ABB RobotStudio station: Eksamens.rspag

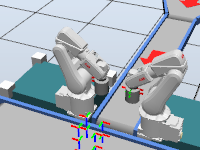
--- station ---
Station Eksamens (saved by RobotStudio 7.0.8746.631)
Controller Virtual_controller, task T_ROB3: task frame (RAPID world) sits at (-5805.06, 703.5, 890) mm, rotated rx 0 ry 0 rz -90 deg in the station
Controller Virtual_controller, task T_ROB2: task frame (RAPID world) sits at (-5805.06, 703.5, 890) mm, rotated rx 0 ry 0 rz -90 deg in the station
Controller Virtual_controller, task T_ROB1: task frame (RAPID world) sits at (-5805.06, 703.5, 890) mm, rotated rx 0 ry 0 rz -90 deg in the station
Controller Virtual_controller
  mechanical unit ROB_1: IRB120_3_58__01_2, 6 joints, base frame (83.5, -144.94, 0) mm
  mechanical unit ROB_2: IRB2600_20_165_C_01_2, 6 joints, base frame (1331.39, 3332.7, 0) mm, rotated rx 0 ry 0 rz 180 deg
  mechanical unit ROB_3: IRB120_3_58__01_3, 6 joints, base frame (643.5, -144.94, 0) mm, rotated rx 0 ry 0 rz 180 deg
Layout (positions relative to the parent item):
  - Sorter_kasser [graphiccomponentgroup]
    - Assemblies [graphiccomponentgroup]
      - Section1 [graphiccomponentgroup]
        - ABB_IRC5_ctrl [graphiccomponentgroup]
          - ABB_IRC5_ctrl_1 [graphiccomponentgroup]
            - Mesh0 [part]
        - Conveyor__Straight_ [graphiccomponentgroup]
          - CONVEYOR1 [graphiccomponentgroup]
            - Mesh1 [part]
            - Mesh2 [part]
            - Mesh3 [part]
          - CONVEYOR2 [graphiccomponentgroup]
            - Mesh4 [part]
            - Mesh5 [part]
            - Mesh6 [part]
          - CONVEYOR3 [graphiccomponentgroup]
            - Mesh7 [part]
            - Mesh8 [part]
            - Mesh9 [part]
          - CONVEYOR4 [graphiccomponentgroup]
            - Mesh10 [part]
            - Mesh11 [part]
            - Mesh12 [part]
          - CONVEYOR5 [graphiccomponentgroup]
            - Mesh13 [part]
            - Mesh14 [part]
            - Mesh15 [part]
          - CONVEYOR6 [graphiccomponentgroup]
            - Mesh16 [part]
            - Mesh17 [part]
            - Mesh18 [part]
          - CONVEYOR7 [graphiccomponentgroup]
            - Mesh19 [part]
            - Mesh20 [part]
            - Mesh21 [part]
        - Cube [graphiccomponentgroup]
          - Cube1 [graphiccomponentgroup]
            - Mesh22 [part]
            - Mesh23 [part]
            - Mesh24 [part]
            - Mesh25 [part]
            - Mesh26 [part]
          - Cube2 [graphiccomponentgroup]
            - Mesh27 [part]
            - Mesh28 [part]
            - Mesh29 [part]
            - Mesh30 [part]
            - Mesh31 [part]
          - Cube3 [graphiccomponentgroup]
            - Mesh32 [part]
            - Mesh33 [part]
            - Mesh34 [part]
            - Mesh35 [part]
            - Mesh36 [part]
        - Eater [graphiccomponentgroup]
          - EATER1 [graphiccomponentgroup]
            - Mesh37 [part]
        - Display [graphiccomponentgroup]
          - EaterSmall [graphiccomponentgroup]
            - Mesh38 [part]
            - Mesh39 [part]
            - Mesh40 [part]
            - Mesh41 [part]
            - Mesh42 [part]
            - Mesh43 [part]
            - Mesh44 [part]
            - Mesh45 [part]
            - Mesh46 [part]
            - Mesh47 [part]
            - Mesh48 [part]
        - Feeder [graphiccomponentgroup]
          - FEEDER1 [graphiccomponentgroup]
            - Mesh49 [part]
            - Mesh50 [part]
          - FEEDER2 [graphiccomponentgroup]
            - Mesh51 [part]
            - Mesh52 [part]
          - FEEDER3 [graphiccomponentgroup]
            - Mesh53 [part]
            - Mesh54 [part]
        - Scale [graphiccomponentgroup]
          - Scale_Weight [graphiccomponentgroup]
            - Mesh55 [part]
            - Mesh56 [part]
            - Mesh57 [part]
            - Mesh58 [part]
          - Scale_Weight1 [graphiccomponentgroup]
            - Mesh59 [part]
            - Mesh60 [part]
            - Mesh61 [part]
            - Mesh62 [part]
          - Scale_Weight2 [graphiccomponentgroup]
            - Mesh63 [part]
            - Mesh64 [part]
            - Mesh65 [part]
            - Mesh66 [part]
        - Text [graphiccomponentgroup]
          - Text1 [graphiccomponentgroup]
            - Mesh67 [part]
    - Motors [graphiccomponentgroup]
      - Surface [graphiccomponentgroup]
        - MOTOR1 [graphiccomponentgroup]
          - Mesh75 [part]
          - Mesh76 [part]
          - Mesh77 [part]
          - Mesh78 [part]
        - MOTOR6 [graphiccomponentgroup]
          - Mesh79 [part]
        - MOTOR8 [graphiccomponentgroup]
          - Mesh80 [part]
        - MOTOR9 [graphiccomponentgroup]
          - Mesh81 [part]
    - Loads [graphiccomponentgroup]
      - Mesh68 [part]
      - Mesh69 [part]
      - Mesh70 [part]
      - Mesh71 [part]
      - Mesh72 [part]
      - Mesh73 [part]
      - Mesh74 [part]
  - IRB120_3_58__01_2 [mechanism, from Robots\IRB120_3_58_G_01.rslib] at (-5950, 620, 890) mm, rotated rx 0 ry 0 rz -90 deg; joint values [-0.0062, -0.4744, 1.1199, 0, 0.9253, -0.0062] (rad or m)
  - IRB2600_20_165_C_01_2 [mechanism, from Robots\IRB2600_20_165_C_01.rslib] at (-2472.36, -627.89, 890) mm, rotated rx 0 ry 0 rz 90 deg; joint values [0, 0.2407, 0.4991, 6.2832, 0.831, 0] (rad or m)
  - IRB120_3_58__01_3 [mechanism, from Robots\IRB120_3_58_G_01.rslib] at (-5950, 60, 890) mm, rotated rx 0 ry 0 rz 90 deg; joint values [0.006, -0.4425, 1.1015, 0, 0.9118, 0.006] (rad or m)
  - GripperStackerRight [mechanism] at (-5951, 460, 1222.41) mm, rotated rx 180 ry 0 rz 90 deg
      TCP GripperStackerRight at (0, 0, 30) mm
      links: SimpleGripper
  - GripperStackerLeft [mechanism] at (-5951, 226, 1222.41) mm, rotated rx 180 ry 0 rz -90 deg
      TCP GripperStackerLeft at (0, 0, 30) mm
      links: SimpleGripper
  - GripperSorter [mechanism] at (-2472.36, 353.71, 1478.82) mm, rotated rx 180 ry 0 rz -90 deg
      TCP GripperSorter at (0, 0, 30) mm
      links: SimpleGripper
Attachment: GripperStackerRight is attached to IRB120_3_58__01_2 / Link6
Attachment: GripperStackerLeft is attached to IRB120_3_58__01_3 / Link6
Attachment: GripperSorter is attached to IRB2600_20_165_C_01_2 / Link6

--- Backups/Virtual_controller/RAPID/TASK1/PROGMOD/CalibData.mod ---
MODULE CalibData
	PERS tooldata GripperStackerRight:=[TRUE,[[0,0,30],[1,0,0,0]],[1,[0,0,1],[1,0,0,0],0,0,0]];
ENDMODULE

--- Backups/Virtual_controller/RAPID/TASK1/PROGMOD/Module1.mod ---
MODULE Module1
    CONST robtarget Right22:=[[305.5,-625.945,302.406],[0,0,1,0],[-1,0,-1,0],[9E+09,9E+09,9E+09,9E+09,9E+09,9E+09]];
    CONST robtarget HomeRight:=[[243.5,-145.945,302.406],[0,0,1,0],[-1,-1,-1,0],[9E+09,9E+09,9E+09,9E+09,9E+09,9E+09]];
    CONST robtarget PickRight:=[[360.5,88.055,133.879],[0,0,1,0],[0,0,0,0],[9E+09,9E+09,9E+09,9E+09,9E+09,9E+09]];
    CONST robtarget Right11:=[[305.5,-515.945,197.406],[0,0,1,0],[-1,0,-1,0],[9E+09,9E+09,9E+09,9E+09,9E+09,9E+09]];
    CONST robtarget Right12:=[[305.5,-625.945,197.406],[0,0,1,0],[-1,0,-1,0],[9E+09,9E+09,9E+09,9E+09,9E+09,9E+09]];
    CONST robtarget Right21:=[[305.5,-515.945,302.406],[0,0,1,0],[-1,0,-1,0],[9E+09,9E+09,9E+09,9E+09,9E+09,9E+09]];

    VAR intnum stackCount := 0;
    !***********************************************************
    !
    ! Module:  Right Stacker robot
    !
    ! Description:
    !   <Insert description here>
    !
    ! Author: madsw
    ! Version: 1.0
    !
    !***********************************************************
    PROC main()
        MoveJ HomeRight, v5000, z100, tool0;
        ! Move when There is and object and Left arm is not in the way.
        IF diStackerRightPick = 1 THEN
            MoveJ PickRight, v5000, z100, tool0;
            MoveJ HomeRight, v5000, z100, tool0;

        ENDIF
    ENDPROC
ENDMODULE

--- Backups/Virtual_controller/RAPID/TASK2/PROGMOD/CalibData.mod ---
MODULE CalibData
	PERS tooldata GripperSorter:=[TRUE,[[0,0,30],[1,0,0,0]],[1,[0,0,1],[1,0,0,0],0,0,0]];
ENDMODULE

--- Backups/Virtual_controller/RAPID/TASK2/PROGMOD/Module1.mod ---
MODULE Module1
    !***********************************************************
    !
    ! Module:  Sorter robot
    !
    ! Description:
    !   <Insert description here>
    !
    ! Author: madsw
    ! Version: 1.0
    !
    !***********************************************************
    PROC main()
        !Add your code here
    ENDPROC
ENDMODULE

--- Backups/Virtual_controller/RAPID/TASK3/PROGMOD/CalibData.mod ---
MODULE CalibData
    PERS tooldata GripperStackerLeft:=[TRUE,[[0,0,30],[1,0,0,0]],[1,[0,0,1],[1,0,0,0],0,0,0]];
ENDMODULE

--- Backups/Virtual_controller/RAPID/TASK3/PROGMOD/Module1.mod ---
MODULE Module1
	CONST robtarget PickLeft:=[[360.5,88.055,133.879],[0,1,0,0],[-1,0,-1,0],[9E+09,9E+09,9E+09,9E+09,9E+09,9E+09]];
	CONST robtarget HomeLeft:=[[477.5,-145.945,302.406],[0,1,0,0],[0,0,0,0],[9E+09,9E+09,9E+09,9E+09,9E+09,9E+09]];
	CONST robtarget Left11:=[[415.5,-515.945,197.406],[0,1,0,0],[0,0,0,0],[9E+09,9E+09,9E+09,9E+09,9E+09,9E+09]];
	CONST robtarget Left12:=[[415.5,-625.945,197.406],[0,1,0,0],[0,0,0,0],[9E+09,9E+09,9E+09,9E+09,9E+09,9E+09]];
	CONST robtarget Left21:=[[415.5,-515.945,302.406],[0,1,0,0],[0,0,0,0],[9E+09,9E+09,9E+09,9E+09,9E+09,9E+09]];
	CONST robtarget Left22:=[[415.5,-625.945,302.406],[0,1,0,0],[0,0,0,0],[9E+09,9E+09,9E+09,9E+09,9E+09,9E+09]];
    !***********************************************************
    !
    ! Module:  Left Stacker robot
    !
    ! Description:
    !   <Insert description here>
    !
    ! Author: madsw
    ! Version: 1.0
    !
    !***********************************************************
    PROC main()
        !Add your code here
    ENDPROC
ENDMODULE

--- Backups/Virtual_controller/SYSPAR/EIO.cfg ---
EIO:CFG_1.0:6:1::
#
EIO_SIGNAL:

      -Name "diSorterPick" -SignalType "DI" -Access "All"

      -Name "diStackerRightPick" -SignalType "DI" -Access "All"

      -Name "diStackerLeftPick" -SignalType "DI" -Access "All"

      -Name "doStackerRightGripper" -SignalType "DO" -Access "All"

      -Name "doStackerLeftGripper" -SignalType "DO" -Access "All"

      -Name "doSorterGripper" -SignalType "DO" -Access "All"
